// TIA Portal V19 export
DATA_BLOCK "A0302_Manager"   // DB84
// stored: InstanceOfName A0302_Manager_FB, InstanceOfType FB
"A0302_Manager_FB"
   // VAR_INPUT
   //    AreaInterface : "AreaInterface";
   //    DataIn : Struct
   //       SemiAut_Pb : Bool;
   //    END_STRUCT;
   //    CIn : Struct
   //       P5 : Struct
   //          Sollevatori { ExternalAccessible := 'False'; ExternalVisible := 'False'; ExternalWritable := 'False'} : "ValveMachine_COut";
   //          Spintore_Lat : Struct
   //             Spin_Lat1 : Struct
   //                Standstill : Bool;
   //                Rest_CheckNext : Bool;
   //                Work_CheckNext : Bool;
   //                Rest : Bool;
   //                Work : Bool;
   //             END_STRUCT;
   //             Spin_Lat2 : Struct
   //                Standstill : Bool;
   //                Rest_CheckNext : Bool;
   //                Work_CheckNext : Bool;
   //                Rest : Bool;
   //                Work : Bool;
   //             END_STRUCT;
   //          END_STRUCT;
   //          SpintoreLong { ExternalAccessible := 'False'; ExternalVisible := 'False'; ExternalWritable := 'False'} : Struct
   //             Ax : "Positioning_EPOS_Machine_COut";
   //             Ax_Sts : Struct
   //                PosAttesa_Reached : Bool;
   //                PosFineSpinta_Reached : Bool;
   //             END_STRUCT;
   //             Spintore : "ValveMachine_COut";
   //             Vrt : "ValveMachine_COut";
   //             Orz : "ValveMachine_COut";
   //             Sens : Struct
   //                FTC_FuoriIngombro : Bool;
   //             END_STRUCT;
   //          END_STRUCT;
   //       END_STRUCT;
   //       Bordatrice : Struct
   //          Ax : "Positioning_EPOS_Machine_COut";
   //          Sts : Struct
   //             PosTargetEnable : Bool;
   //             PosTarget_Reached : Bool;
   //             In_W_Pos : Bool;
   //             AtRest : Bool;
   //          END_STRUCT;
   //          Sens : Struct
   //             FTC_Ingresso : Bool;
   //             FTC_Uscita : Bool;
   //          END_STRUCT;
   //       END_STRUCT;
   //       Rulliera { ExternalAccessible := 'False'; ExternalVisible := 'False'; ExternalWritable := 'False'} : Struct
   //          Ax_1 : "SpeedMachine_COut";
   //          Ax_2 : "SpeedMachine_COut";
   //          Centraggio : "ValveMachine_COut";
   //          Sollevamento : "ValveMachine_COut";
   //          Coda : Struct
   //             Sens : Struct
   //                FTC_Rall : Bool;
   //                FTC_Prox_Ing : Bool;
   //             END_STRUCT;
   //          END_STRUCT;
   //          Centro : Struct
   //             Sens : Struct
   //                FTC_Centrale : Bool;
   //             END_STRUCT;
   //          END_STRUCT;
   //       END_STRUCT;
   //       CarroPareggCoda { ExternalAccessible := 'False'; ExternalVisible := 'False'; ExternalWritable := 'False'} : Struct
   //          Ax_InWPos : Bool;
   //          Ax : "Positioning_DOL_Machine_COut";
   //          Bloccaggio : "ValveMachine_COut";
   //          BattutaVerticale : "ValveMachine_COut";
   //          PareggiatoreLong : "ValveMachine_COut";
   //          Sens : Struct
   //             FTC_Ingombro_Ing : Bool;
   //             FTC_Ingombro_Out : Bool;
   //             PresenzaMat : Bool;
   //             PosPareggLong : Struct
   //                Value : LReal;
   //                CheckMeasure : Bool;
   //                Standstill : Bool;
   //             END_STRUCT;
   //          END_STRUCT;
   //       END_STRUCT;
   //       CarroPareggTesta { ExternalAccessible := 'False'; ExternalVisible := 'False'; ExternalWritable := 'False'} : Struct
   //          Ax_InWPos : Bool;
   //          Ax : "Positioning_DOL_Machine_COut";
   //          Bloccaggio : "ValveMachine_COut";
   //          Centraggio : "ValveMachine_COut";
   //          Sollevatore : "ValveMachine_COut";
   //          Sens : Struct
   //             FTC_Ingombro_Ing : Bool;
   //             FTC_Prox_Ls : Bool;
   //             PresenzaMat : Bool;
   //          END_STRUCT;
   //       END_STRUCT;
   //       Manipolatori : Struct
   //          Testa : Struct
   //             Ax : "Positioning_EPOS_Machine_COut";
   //             Sollevatore : "ValveMachine_COut";
   //             Magnete : "ValveMachine_COut";
   //          END_STRUCT;
   //          Coda : Struct
   //             Ax : "Positioning_EPOS_Machine_COut";
   //             Sollevatore : "ValveMachine_COut";
   //             Magnete : "ValveMachine_COut";
   //          END_STRUCT;
   //          InPos_Prelievo : Bool;
   //          InPos_BancoScarto : Bool;
   //          InPos_BancoA0303 : Bool;
   //       END_STRUCT;
   //       Spalle : Struct
   //          Coda : Struct
   //             Ax : "Positioning_DOL_Machine_COut";
   //          END_STRUCT;
   //          Testa : Struct
   //             Ax : "Positioning_DOL_Machine_COut";
   //          END_STRUCT;
   //       END_STRUCT;
   //       Banco_A0303 : Struct
   //          ReadyToRecive : Bool;
   //       END_STRUCT;
   //       ProdManager : "Prod_Beam_Ctrl";
   //    END_STRUCT;
   // END_VAR
   // VAR_OUTPUT
   //    MachineInterface : "MachineInterface";
   //    COut : Struct
   //       HU : Struct
   //          EnableStopDoorOpeningReq : Bool;
   //          EnableStopInPhase : Bool;
   //          EnableStopProgrammed : Bool;
   //          Control_ON : Bool;
   //          Rest : Bool;
   //          Work : Bool;
   //       END_STRUCT;
   //       SpintoreLong : Struct
   //          EnableStopDoorOpeningReq : Bool;
   //          EnableStopInPhase : Bool;
   //          EnableStopProgrammed : Bool;
   //          Control_ON : Bool;
   //          REST_Req : Bool;
   //          WORK_Req : Bool;
   //          Rest : Bool;
   //          Work : Bool;
   //       END_STRUCT;
   //       Bordatrice : Struct
   //          Ax : "Positioning_EPOS_Machine_Manager";
   //          Sts : Struct
   //             PosTarget_Reached : Bool;
   //             AtRest : Bool;
   //          END_STRUCT;
   //          DataOut : "Positioning_EPOS_Machine_DataOut";
   //          Rest_Req : Bool;
   //          Work_Req : Bool;
   //       END_STRUCT;
   //       Rulliera : Struct
   //          Ax_1 : "SpeedMachine_CIn_Manager";
   //          Ax_2 : "SpeedMachine_CIn_Manager";
   //          Centratori : Struct
   //             Sollevamento : "ValveMachine_Manager";
   //             Centraggio : "ValveMachine_Manager";
   //          END_STRUCT;
   //          Ax_1_Frw_Req : Bool;
   //          Ax_1_Brw_Req : Bool;
   //          Ax_2_Frw_Req : Bool;
   //          Ax_2_Brw_Req : Bool;
   //       END_STRUCT;
   //       CarroPareggCoda : Struct
   //          EnableStopDoorOpeningReq : Bool;
   //          EnableStopInPhase : Bool;
   //          EnableStopProgrammed : Bool;
   //          Control_ON : Bool;
   //          MoveToPos : Bool;
   //          Pos : LReal;
   //          Speed : LReal;
   //          Bloccaggio : Struct
   //             Rest : Bool;
   //             Work : Bool;
   //          END_STRUCT;
   //          BattutaVrt : Struct
   //             Rest : Bool;
   //             Work : Bool;
   //          END_STRUCT;
   //          PareggLong : Struct
   //             Rest : Bool;
   //             Work : Bool;
   //          END_STRUCT;
   //       END_STRUCT;
   //       CarroPareggTesta : Struct
   //          EnableStopDoorOpeningReq : Bool;
   //          EnableStopInPhase : Bool;
   //          EnableStopProgrammed : Bool;
   //          Control_ON : Bool;
   //          MoveToPos : Bool;
   //          Pos : LReal;
   //          Speed : LReal;
   //          Bloccaggio : "OP_PB";
   //          Sollevamento : "OP_PB";
   //          Centraggio : "OP_PB";
   //       END_STRUCT;
   //       Manipolatori : Struct
   //          Ax : Struct
   //             EnableStopDoorOpeningReq : Bool;
   //             EnableStopInPhase : Bool;
   //             EnableStopProgrammed : Bool;
   //             Control_ON : Bool;
   //             MoveToPos : Bool;
   //             Pos : LReal;
   //             Vel : LReal;
   //             Acc : LReal;
   //             Dec : LReal;
   //          END_STRUCT;
   //          Sollevatori : "OP_PB";
   //          Magneti : "OP_PB";
   //       END_STRUCT;
   //    END_STRUCT;
   // END_VAR
   // VAR_IN_OUT
   //    Par : Struct
   //       CarroPareggCoda : Struct
   //          Delay_StartMove : Time;
   //          Preset : LReal;
   //       END_STRUCT;
   //       CarroPareggTesta : Struct
   //          Delay_StartMove : Time;
   //          Preset : LReal;
   //       END_STRUCT;
   //       Cremaliera : Struct
   //          Modulo : LReal;
   //          Passo : LReal;
   //       END_STRUCT;
   //    END_STRUCT;
   // END_VAR
   // VAR
   //    Alarm : Struct
   //       Qlty_Unknow : Bool;
   //       ToCheckList_Full : Bool;
   //       WrongReadPz_ManipBasso : Bool;
   //       Pz_NonPareggiabile : Bool;
   //       STOP_FineTurno : Bool;
   //       STOP_End_Of_Proroduction : Bool;
   //       STOP_ControlloQualita : Bool;
   //    END_STRUCT;
   //    Warning : Struct
   //       CheckBancoAccumulo : Bool;
   //    END_STRUCT;
   //    Sts : Struct
   //       SemiAut : Struct
   //          ON : Bool;
   //          Request : Bool;
   //          MaterialFrw : Bool;
   //       END_STRUCT;
   //       CarroPareggTesta : Struct
   //          InCyclePos : Bool;
   //       END_STRUCT;
   //       CarroPareggCoda : Struct
   //          InCyclePos : Bool;
   //       END_STRUCT;
   //       Attrezzamento : Struct
   //          Ready : Bool;
   //          FindNewID : Bool;
   //          RequestNewPosition : Bool;
   //          OLD_OID : DInt;
   //       END_STRUCT;
   //       BTrk : Struct
   //          A0302Exit_Actual_O_ID : DInt;
   //          BLen_Paregg : Real;
   //          Last_Misure1Paregg : Real;
   //          Last_Misure2Paregg : Real;
   //          A0302Entry_Absence : Bool;
   //          A0302Exit_Absence : Bool;
   //          ZoneA0302Entry_Empty : Bool;
   //          ZoneA0302Exit_Empty : Bool;
   //          A0302_CheckBancoAccumulo : Bool;
   //          Waiting_A0302_Recive : Bool;
   //       END_STRUCT;
   //       AlarmsPresence : Bool;
   //       WarningsPresence : Bool;
   //       IsStandstill : Bool;
   //    END_STRUCT;
   //    Ctrl : Struct
   //       Stop : Bool;
   //       TRK : Struct
   //          BTrk : Struct
   //             "P5.1_To_LongPosAttesa" : Bool;
   //             "P5.2_LongPosAttesa_TO_Spintore" : Bool;
   //             "P5.2_Spintore_TO_ExitA031" : Bool;
   //             "P5.2_ExitA031_To_IngBord" : Bool;
   //             "P5.2_Ax_MoveToPosAttesa" : Bool;
   //             "P5.2_Ax_PreparingPosAttesa" : Bool;
   //             "P5.2_Ax_MoveToPosSpinta" : Bool;
   //             SpinBord_In_To_Bord_In : Bool;
   //             Bordatrice_In_To_Out : Bool;
   //             Bordatrice_Out_To_PareggCodaUp : Bool;
   //             Bordatrice_Out_To_PareggCodaDown : Bool;
   //             Rulliera_Start_Brw : Bool;
   //             Rulliera_Ax_1_Start_Frw : Bool;
   //             Rulliera_Ax_2_Start_Frw : Bool;
   //             RulliereVode : Bool;
   //             PCodaDown_TO_Rulli_PCodaDown : Bool;
   //             PCodaDown_TO_RALL_Rulli_PCodaDown : Bool;
   //             PCodaDown_TO_STOP_PCodaDown : Bool;
   //             STOP_PCodaDown_TO_PCoda_Up : Bool;
   //             "PareggCodaUp_To_Rull-PrimaPareggCodaAltro" : Bool;
   //             PCoda_Up_TO_PCoda_UP_S3 : Bool;
   //             PCoda_UP_S3_TO_PCoda_UP_S4 : Bool;
   //             PCoda_UP_S4_TO_PCoda_DownCnd : Bool;
   //             PCoda_Beam_TO_PTesta : Bool;
   //             Beam_TO_Stop_PTesta : Bool;
   //             "Stop_PTesta_TO_Rull-Centratori" : Bool;
   //             "Rull-Centratori_TO_Cnd_PareggCoda" : Bool;
   //             Cnd_PareggCoda_TO_Pareggiato : Bool;
   //             Check_Tolleranza_BLen_Qlty : Bool;
   //             Pareggiato_TO_PresaBasso : Bool;
   //             PresaBasso_TO_PresaAlto : Bool;
   //             PresaAlto_To_CheckOut_BadQlty : Bool;
   //             CheckOut_BadQlty_UP_MoveToPos : Bool;
   //             PresaAlto_To_CheckOut_GoodQlty : Bool;
   //             CheckOut_GoodQlty_UP_MoveToPos : Bool;
   //             CheckOut_BadQlty_UP_To_DOWN : Bool;
   //             CheckOut_BadQlty_DOWN_To_Sgancia : Bool;
   //             CheckOut_GoodQlty_UP_To_DOWN : Bool;
   //             CheckOut_GoodQlty_DOWN_To_Sgancia : Bool;
   //             Manipolatori_Return_ToPrelievo : Bool;
   //          END_STRUCT;
   //          BTrk_ToCheck : Struct
   //             ClearList : Bool;
   //             QtyClear_RetVal : Bool;
   //             Prelievo_RecondGood : Bool;
   //             RecG_InPos_Centraggio : Bool;
   //             RegG_InPos_ReadyPickUp : Bool;
   //          END_STRUCT;
   //       END_STRUCT;
   //       SpintoreLong : Struct
   //          Rest : Bool;
   //          Work : Bool;
   //          MoveAttesaDisable : Bool;
   //       END_STRUCT;
   //       Bordatrice : Struct
   //          Run : Bool;
   //       END_STRUCT;
   //       Rulliera : Struct
   //          Ax_1_Vel_Bord : Bool;
   //          Ax_2_Vel_Bord : Bool;
   //          Ax_1_Lenta_CarroCoda : Bool;
   //          Ax_1_2_Vel_CarroTesta : Bool;
   //          Ax_1_2_Vel_ZeroTesta : Bool;
   //          Ax_1_2_Vel_Appoggio : Bool;
   //          Ax_1_2_End_VelZero : Bool;
   //          Ax_2_MemoRall : Bool;
   //          SP_TimeMemoRall : Time;
   //          TON_RitardoRallenta : IEC_TIMER;
   //          Centraggio : Struct
   //             Rest : Bool;
   //             Work : Bool;
   //          END_STRUCT;
   //          Sollevamento : Struct
   //             Rest : Bool;
   //             Work : Bool;
   //          END_STRUCT;
   //       END_STRUCT;
   //       CarroPareggCoda : Struct
   //          Ax : Struct
   //             MoveToPos : Bool;
   //             Pos : LReal;
   //          END_STRUCT;
   //          Bloccaggio : Struct
   //             Rest : Bool;
   //             Work : Bool;
   //          END_STRUCT;
   //          BattutaVerticale : Struct
   //             Rest : Bool;
   //             Work : Bool;
   //          END_STRUCT;
   //          PareggiatoreLong : Struct
   //             Rest : Bool;
   //             Work : Bool;
   //          END_STRUCT;
   //          MisuraPzPareggiato : Bool;
   //       END_STRUCT;
   //       CarroPareggTesta : Struct
   //          Ax : Struct
   //             MoveToPos : Bool;
   //             Pos : LReal;
   //          END_STRUCT;
   //          Bloccaggio : Struct
   //             Rest : Bool;
   //             Work : Bool;
   //          END_STRUCT;
   //          Sollevatore : Struct
   //             Rest : Bool;
   //             Work : Bool;
   //          END_STRUCT;
   //          Centraggio : Struct
   //             Rest : Bool;
   //             Work : Bool;
   //          END_STRUCT;
   //       END_STRUCT;
   //       Manipolatori : Struct
   //          Ax : Struct
   //             MoveToPos : Bool;
   //             Pos : LReal;
   //          END_STRUCT;
   //          Sollevatori : Struct
   //             Rest : Bool;
   //             Work : Bool;
   //          END_STRUCT;
   //          Magneti : Struct
   //             Rest : Bool;
   //             Work : Bool;
   //          END_STRUCT;
   //       END_STRUCT;
   //    END_STRUCT;
   //    HMI : Struct
   //       PlsClear_ListToCheck : Bool;
   //    END_STRUCT;
   //    BTrk_A0302_Exit_Item : Struct
   //       BLean : Real;
   //       W_A : Real;
   //       Tol_Max : Real;
   //       Tol_Min : Real;
   //       Good { ExternalAccessible := 'False'; ExternalVisible := 'False'; ExternalWritable := 'False'} : Bool;
   //       ToCheckLen { ExternalAccessible := 'False'; ExternalVisible := 'False'; ExternalWritable := 'False'} : Bool;
   //    END_STRUCT;
   //    BTrk_ListToCheck : Struct
   //       Recond : Struct
   //          Found : Bool;
   //          Nr_B : Int;
   //       END_STRUCT;
   //    END_STRUCT;
   //    OffsetCarri : Struct
   //       DaSpallaTesta : LReal;
   //       DaSpallaCoda : LReal;
   //    END_STRUCT;
   //    CarroTesta : Struct
   //       RimanenzaPos : LReal;
   //       PassoReq : LReal;
   //       PosBattutePz : LReal;
   //       SemiBeamLen : LReal;
   //       NrPassiReq : LReal;
   //    END_STRUCT;
   //    CarroCoda : Struct
   //       RimanenzaPos : LReal;
   //       PassoReq : LReal;
   //       PosBattutePz : LReal;
   //       SemiBeamLen : LReal;
   //       NrPassiReq : LReal;
   //    END_STRUCT;
   //    TON_AlarmWrongReadPz_Manip : IEC_TIMER;
   //    TON_Alarm_FTC_CarroCodaOut { S7_SetPoint := 'True'} : IEC_TIMER;
   //    TON_Stop { S7_SetPoint := 'True'} : IEC_TIMER;
   // END_VAR
BEGIN
END_DATA_BLOCK
